{attribute addProperty BoxType "EL5101-0000-1019"}
{attribute addProperty Id "Enable_latch_CAT %Q*BOOL811Enable_latch_extern_on_positive_edgeAT %Q*BOOL812Set_counterAT %Q*BOOL813Enable_latch_extern_on_negative_edgeAT %Q*BOOL814Set_counter_valueAT %Q*UINT16217"}
{attribute addProperty CRC "2917873719"}
{attribute addProperty SizeInBites "48"}
{attribute addProperty SizeInBytes "6"}
TYPE ENC_Control_compact_ADEB3837 :
STRUCT
	{attribute addProperty Name "Enable_latch_C"}
	Enable_latch_C AT %Q* : BOOL;
	{attribute addProperty Name "Enable_latch_extern_on_positive_edge"}
	Enable_latch_extern_on_positive_edge AT %Q* : BOOL;
	{attribute addProperty Name "Set_counter"}
	Set_counter AT %Q* : BOOL;
	{attribute addProperty Name "Enable_latch_extern_on_negative_edge"}
	Enable_latch_extern_on_negative_edge AT %Q* : BOOL;
	{attribute addProperty Name "Set_counter_value"}
	Set_counter_value AT %Q* : UINT;
END_STRUCT
END_TYPE

(* stored: Version 1.2.0.0, ProductVersion 3.1.4024.9
   DUT ENC_Control_compact_ADEB3837: Id {1db37fb1-d47a-4e38-a33e-a26f83102d3c} *)
